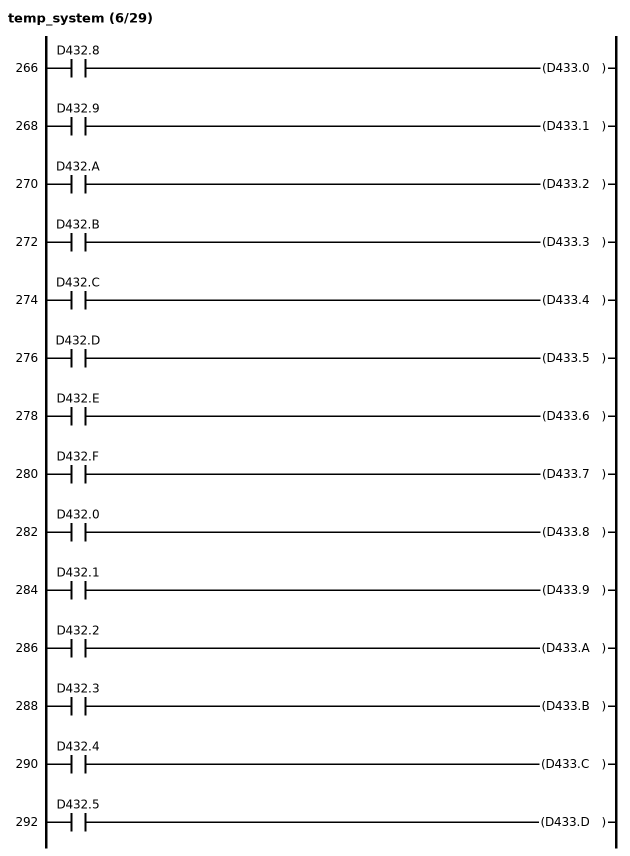
[picture p288: ladder of temp_system, rungs at steps 266 to 292]
266   LD      D432.8
      OUT     D433.0
268   LD      D432.9
      OUT     D433.1
270   LD      D432.A
      OUT     D433.2
272   LD      D432.B
      OUT     D433.3
274   LD      D432.C
      OUT     D433.4
276   LD      D432.D
      OUT     D433.5
278   LD      D432.E
      OUT     D433.6
280   LD      D432.F
      OUT     D433.7
282   LD      D432.0
      OUT     D433.8
284   LD      D432.1
      OUT     D433.9
286   LD      D432.2
      OUT     D433.A
288   LD      D432.3
      OUT     D433.B
290   LD      D432.4
      OUT     D433.C
292   LD      D432.5
      OUT     D433.D
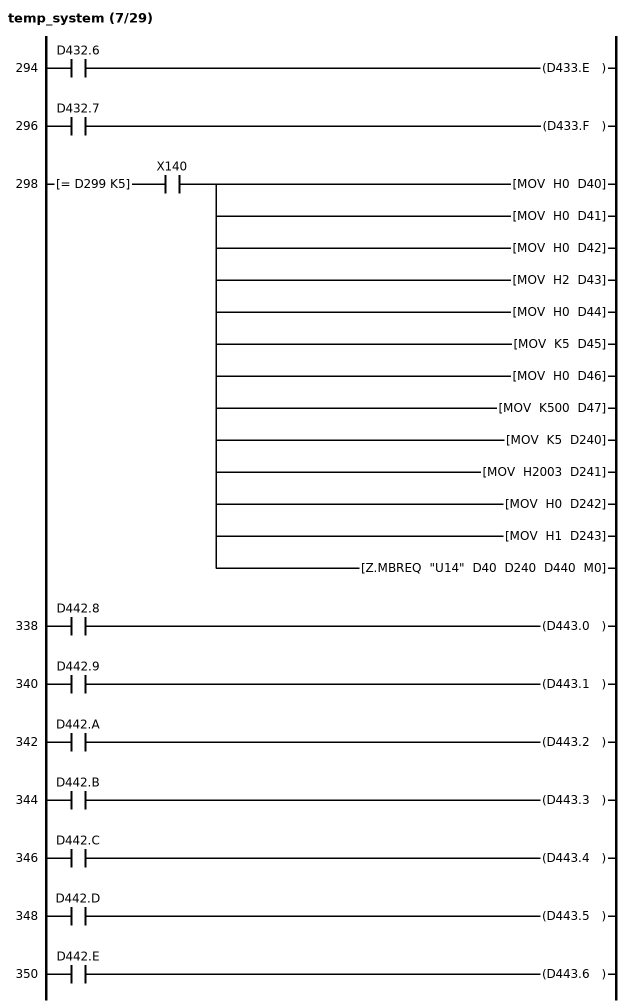
294   LD      D432.6
      OUT     D433.E
296   LD      D432.7
      OUT     D433.F
298   LD=     D299 K5
      AND     X140
      MOV     H0 D40
      MOV     H0 D41
      MOV     H0 D42
      MOV     H2 D43
      MOV     H0 D44
      MOV     K5 D45
      MOV     H0 D46
      MOV     K500 D47
      MOV     K5 D240
      MOV     H2003 D241
      MOV     H0 D242
      MOV     H1 D243
      Z.MBREQ "U14" D40 D240 D440 M0
338   LD      D442.8
      OUT     D443.0
340   LD      D442.9
      OUT     D443.1
342   LD      D442.A
      OUT     D443.2
344   LD      D442.B
      OUT     D443.3
346   LD      D442.C
      OUT     D443.4
348   LD      D442.D
      OUT     D443.5
350   LD      D442.E
      OUT     D443.6
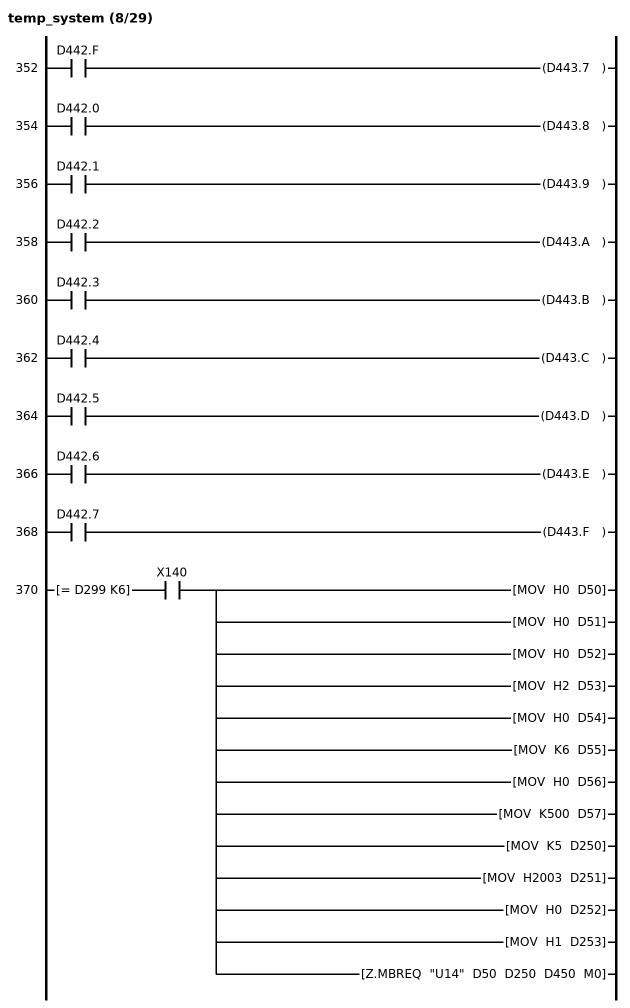
352   LD      D442.F
      OUT     D443.7
354   LD      D442.0
      OUT     D443.8
356   LD      D442.1
      OUT     D443.9
358   LD      D442.2
      OUT     D443.A
360   LD      D442.3
      OUT     D443.B
362   LD      D442.4
      OUT     D443.C
364   LD      D442.5
      OUT     D443.D
366   LD      D442.6
      OUT     D443.E
368   LD      D442.7
      OUT     D443.F
370   LD=     D299 K6
      AND     X140
      MOV     H0 D50
      MOV     H0 D51
      MOV     H0 D52
      MOV     H2 D53
      MOV     H0 D54
      MOV     K6 D55
      MOV     H0 D56
      MOV     K500 D57
      MOV     K5 D250
      MOV     H2003 D251
      MOV     H0 D252
      MOV     H1 D253
      Z.MBREQ "U14" D50 D250 D450 M0
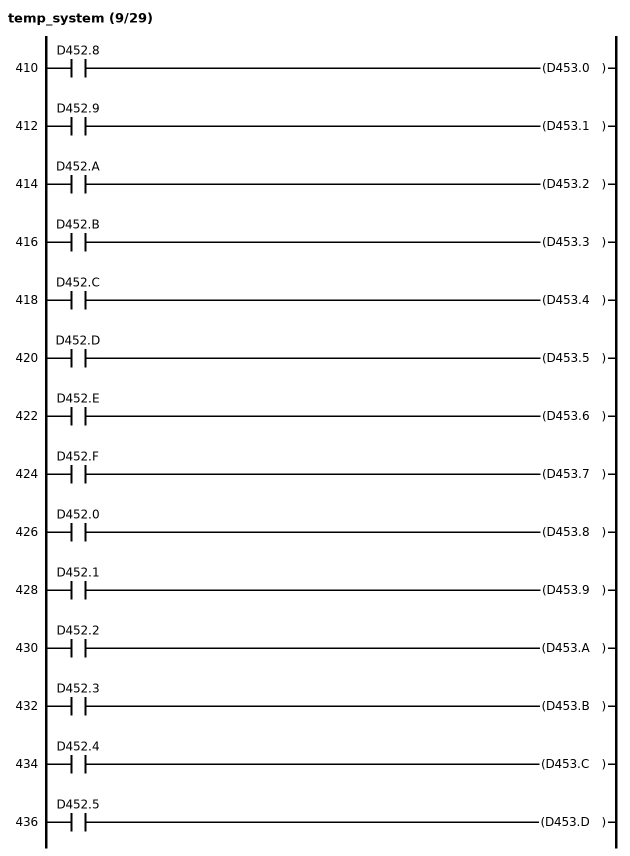
410   LD      D452.8
      OUT     D453.0
412   LD      D452.9
      OUT     D453.1
414   LD      D452.A
      OUT     D453.2
416   LD      D452.B
      OUT     D453.3
418   LD      D452.C
      OUT     D453.4
420   LD      D452.D
      OUT     D453.5
422   LD      D452.E
      OUT     D453.6
424   LD      D452.F
      OUT     D453.7
426   LD      D452.0
      OUT     D453.8
428   LD      D452.1
      OUT     D453.9
430   LD      D452.2
      OUT     D453.A
432   LD      D452.3
      OUT     D453.B
434   LD      D452.4
      OUT     D453.C
436   LD      D452.5
      OUT     D453.D
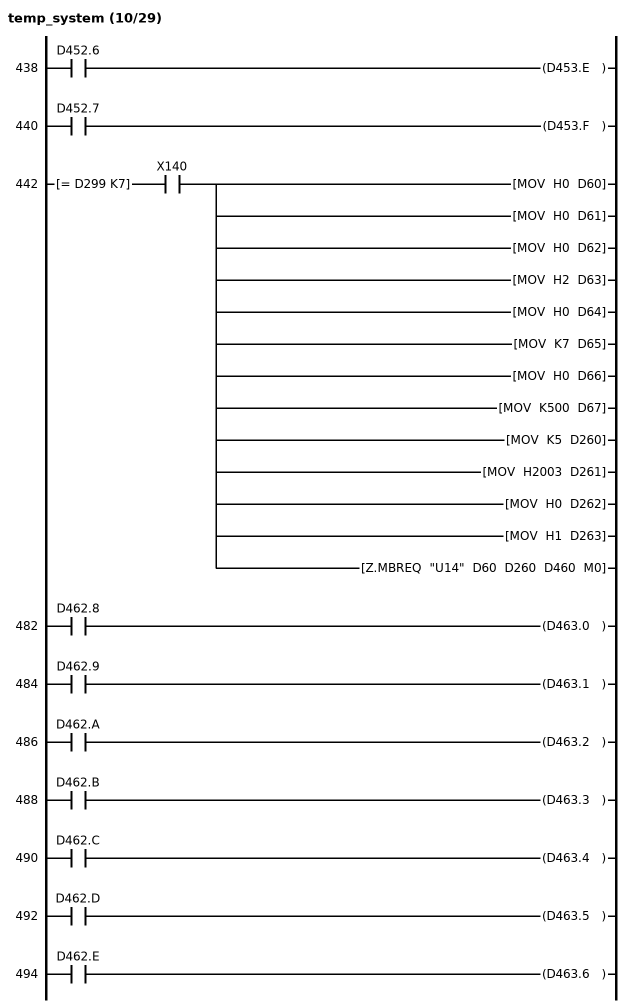
438   LD      D452.6
      OUT     D453.E
440   LD      D452.7
      OUT     D453.F
442   LD=     D299 K7
      AND     X140
      MOV     H0 D60
      MOV     H0 D61
      MOV     H0 D62
      MOV     H2 D63
      MOV     H0 D64
      MOV     K7 D65
      MOV     H0 D66
      MOV     K500 D67
      MOV     K5 D260
      MOV     H2003 D261
      MOV     H0 D262
      MOV     H1 D263
      Z.MBREQ "U14" D60 D260 D460 M0
482   LD      D462.8
      OUT     D463.0
484   LD      D462.9
      OUT     D463.1
486   LD      D462.A
      OUT     D463.2
488   LD      D462.B
      OUT     D463.3
490   LD      D462.C
      OUT     D463.4
492   LD      D462.D
      OUT     D463.5
494   LD      D462.E
      OUT     D463.6
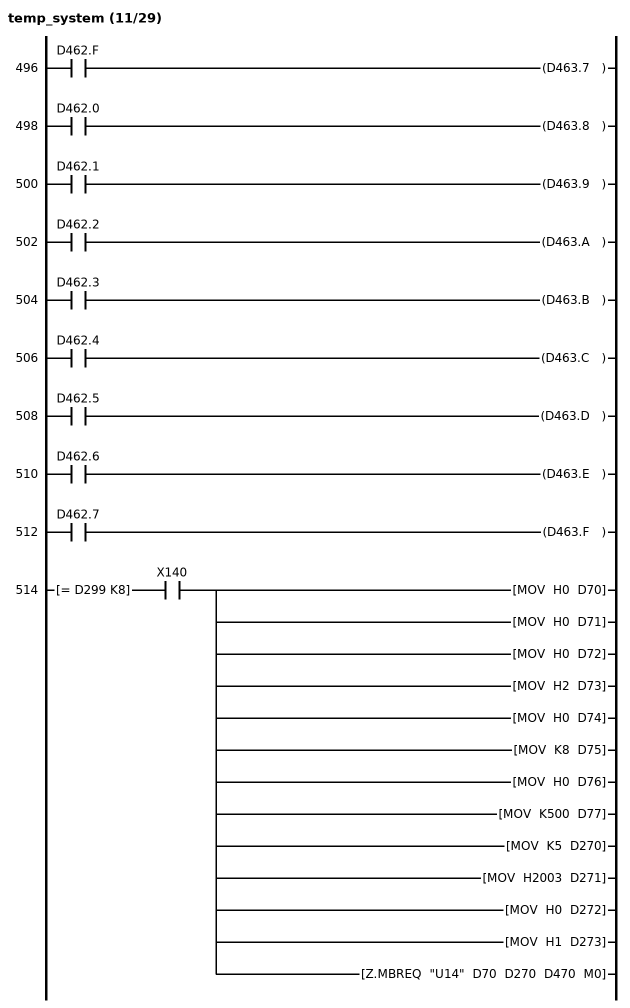
496   LD      D462.F
      OUT     D463.7
498   LD      D462.0
      OUT     D463.8
500   LD      D462.1
      OUT     D463.9
502   LD      D462.2
      OUT     D463.A
504   LD      D462.3
      OUT     D463.B
506   LD      D462.4
      OUT     D463.C
508   LD      D462.5
      OUT     D463.D
510   LD      D462.6
      OUT     D463.E
512   LD      D462.7
      OUT     D463.F
514   LD=     D299 K8
      AND     X140
      MOV     H0 D70
      MOV     H0 D71
      MOV     H0 D72
      MOV     H2 D73
      MOV     H0 D74
      MOV     K8 D75
      MOV     H0 D76
      MOV     K500 D77
      MOV     K5 D270
      MOV     H2003 D271
      MOV     H0 D272
      MOV     H1 D273
      Z.MBREQ "U14" D70 D270 D470 M0
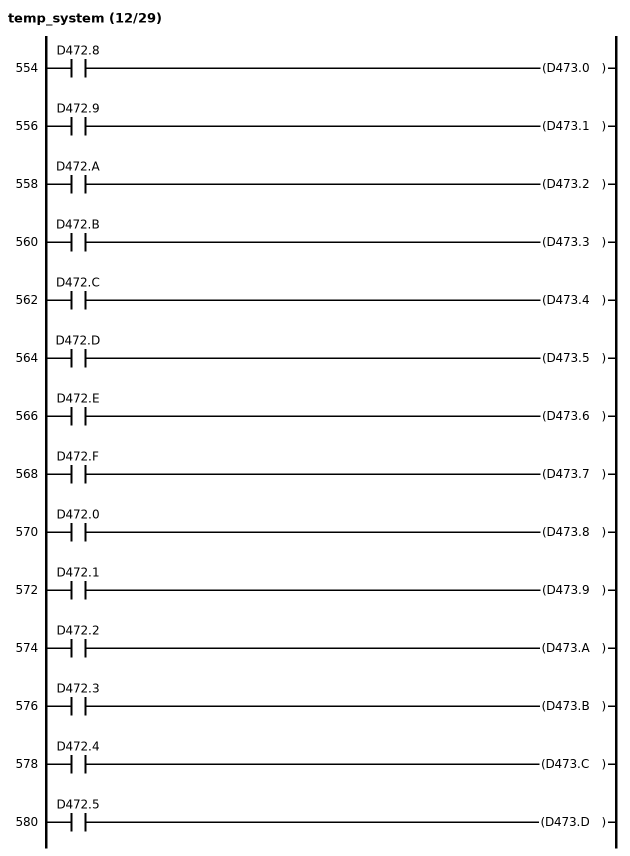
554   LD      D472.8
      OUT     D473.0
556   LD      D472.9
      OUT     D473.1
558   LD      D472.A
      OUT     D473.2
560   LD      D472.B
      OUT     D473.3
562   LD      D472.C
      OUT     D473.4
564   LD      D472.D
      OUT     D473.5
566   LD      D472.E
      OUT     D473.6
568   LD      D472.F
      OUT     D473.7
570   LD      D472.0
      OUT     D473.8
572   LD      D472.1
      OUT     D473.9
574   LD      D472.2
      OUT     D473.A
576   LD      D472.3
      OUT     D473.B
578   LD      D472.4
      OUT     D473.C
580   LD      D472.5
      OUT     D473.D
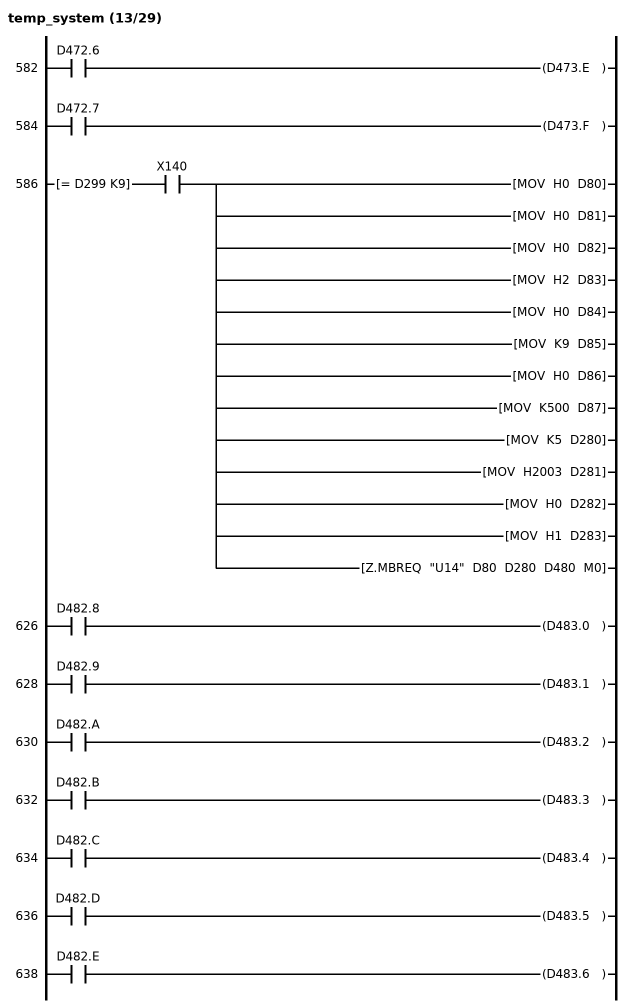
582   LD      D472.6
      OUT     D473.E
584   LD      D472.7
      OUT     D473.F
586   LD=     D299 K9
      AND     X140
      MOV     H0 D80
      MOV     H0 D81
      MOV     H0 D82
      MOV     H2 D83
      MOV     H0 D84
      MOV     K9 D85
      MOV     H0 D86
      MOV     K500 D87
      MOV     K5 D280
      MOV     H2003 D281
      MOV     H0 D282
      MOV     H1 D283
      Z.MBREQ "U14" D80 D280 D480 M0
626   LD      D482.8
      OUT     D483.0
628   LD      D482.9
      OUT     D483.1
630   LD      D482.A
      OUT     D483.2
632   LD      D482.B
      OUT     D483.3
634   LD      D482.C
      OUT     D483.4
636   LD      D482.D
      OUT     D483.5
638   LD      D482.E
      OUT     D483.6
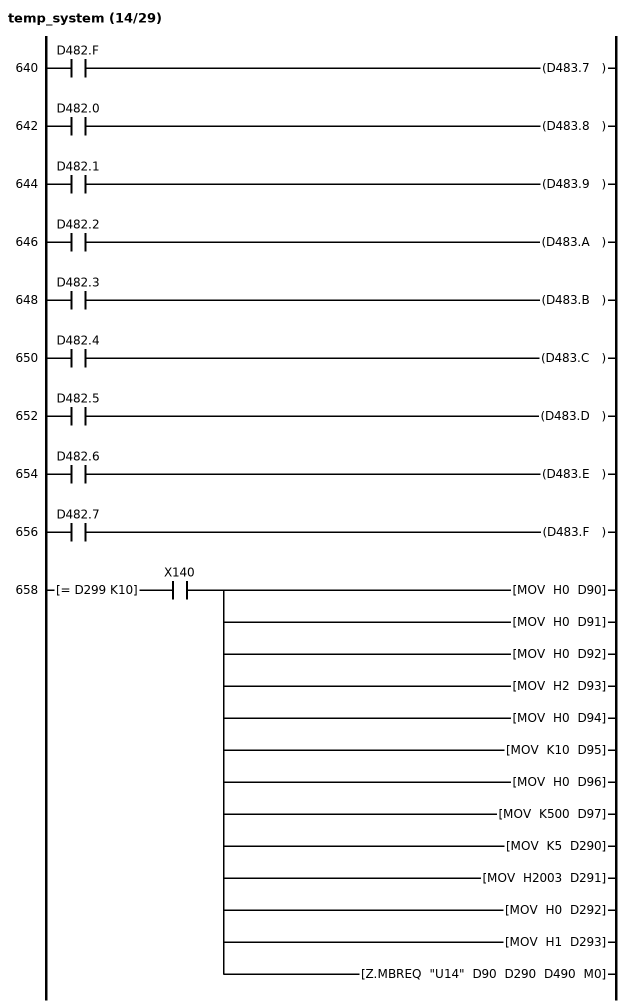
640   LD      D482.F
      OUT     D483.7
642   LD      D482.0
      OUT     D483.8
644   LD      D482.1
      OUT     D483.9
646   LD      D482.2
      OUT     D483.A
648   LD      D482.3
      OUT     D483.B
650   LD      D482.4
      OUT     D483.C
652   LD      D482.5
      OUT     D483.D
654   LD      D482.6
      OUT     D483.E
656   LD      D482.7
      OUT     D483.F
658   LD=     D299 K10
      AND     X140
      MOV     H0 D90
      MOV     H0 D91
      MOV     H0 D92
      MOV     H2 D93
      MOV     H0 D94
      MOV     K10 D95
      MOV     H0 D96
      MOV     K500 D97
      MOV     K5 D290
      MOV     H2003 D291
      MOV     H0 D292
      MOV     H1 D293
      Z.MBREQ "U14" D90 D290 D490 M0
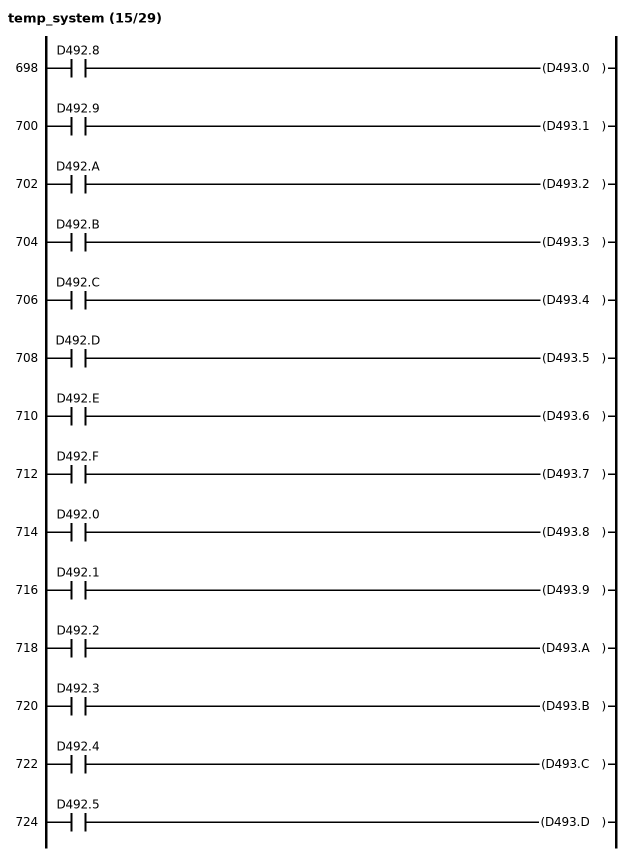
698   LD      D492.8
      OUT     D493.0
700   LD      D492.9
      OUT     D493.1
702   LD      D492.A
      OUT     D493.2
704   LD      D492.B
      OUT     D493.3
706   LD      D492.C
      OUT     D493.4
708   LD      D492.D
      OUT     D493.5
710   LD      D492.E
      OUT     D493.6
712   LD      D492.F
      OUT     D493.7
714   LD      D492.0
      OUT     D493.8
716   LD      D492.1
      OUT     D493.9
718   LD      D492.2
      OUT     D493.A
720   LD      D492.3
      OUT     D493.B
722   LD      D492.4
      OUT     D493.C
724   LD      D492.5
      OUT     D493.D
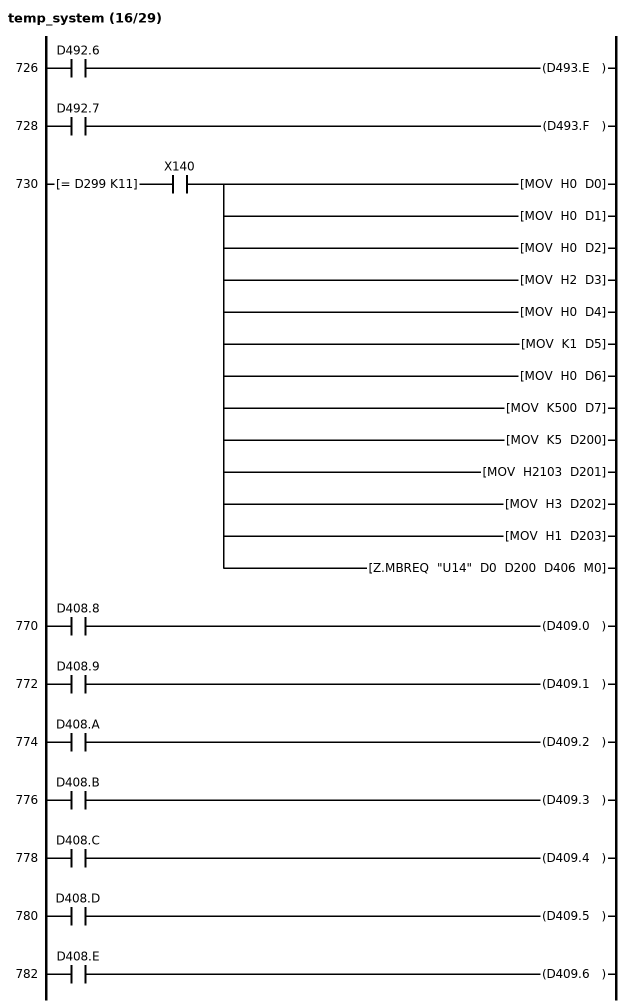
726   LD      D492.6
      OUT     D493.E
728   LD      D492.7
      OUT     D493.F
730   LD=     D299 K11
      AND     X140
      MOV     H0 D0
      MOV     H0 D1
      MOV     H0 D2
      MOV     H2 D3
      MOV     H0 D4
      MOV     K1 D5
      MOV     H0 D6
      MOV     K500 D7
      MOV     K5 D200
      MOV     H2103 D201
      MOV     H3 D202
      MOV     H1 D203
      Z.MBREQ "U14" D0 D200 D406 M0
770   LD      D408.8
      OUT     D409.0
772   LD      D408.9
      OUT     D409.1
774   LD      D408.A
      OUT     D409.2
776   LD      D408.B
      OUT     D409.3
778   LD      D408.C
      OUT     D409.4
780   LD      D408.D
      OUT     D409.5
782   LD      D408.E
      OUT     D409.6
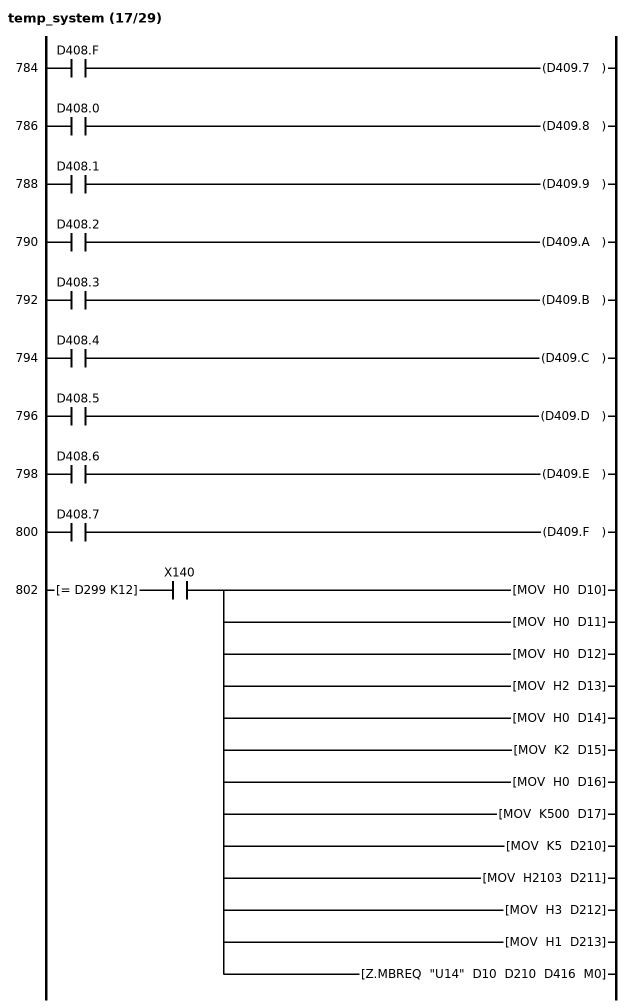
784   LD      D408.F
      OUT     D409.7
786   LD      D408.0
      OUT     D409.8
788   LD      D408.1
      OUT     D409.9
790   LD      D408.2
      OUT     D409.A
792   LD      D408.3
      OUT     D409.B
794   LD      D408.4
      OUT     D409.C
796   LD      D408.5
      OUT     D409.D
798   LD      D408.6
      OUT     D409.E
800   LD      D408.7
      OUT     D409.F
802   LD=     D299 K12
      AND     X140
      MOV     H0 D10
      MOV     H0 D11
      MOV     H0 D12
      MOV     H2 D13
      MOV     H0 D14
      MOV     K2 D15
      MOV     H0 D16
      MOV     K500 D17
      MOV     K5 D210
      MOV     H2103 D211
      MOV     H3 D212
      MOV     H1 D213
      Z.MBREQ "U14" D10 D210 D416 M0
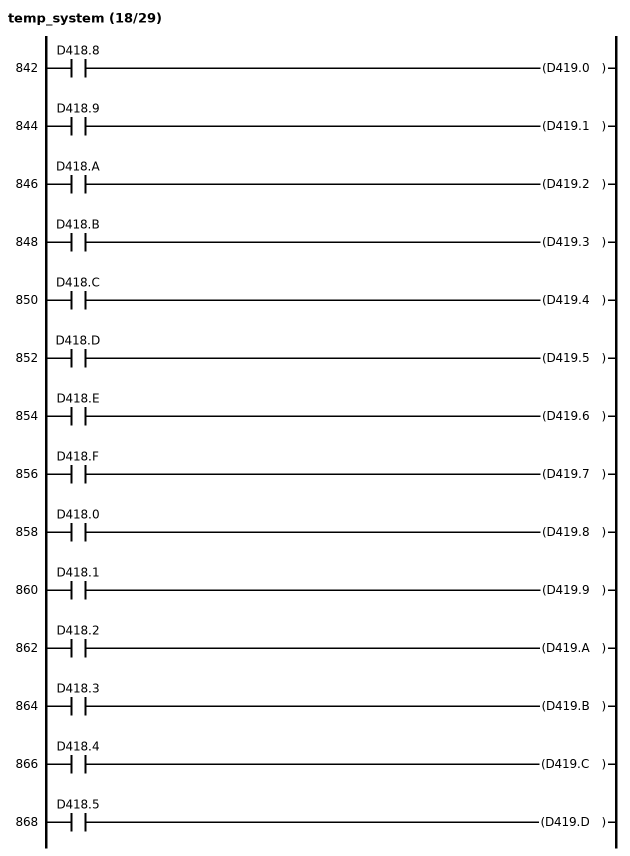
842   LD      D418.8
      OUT     D419.0
844   LD      D418.9
      OUT     D419.1
846   LD      D418.A
      OUT     D419.2
848   LD      D418.B
      OUT     D419.3
850   LD      D418.C
      OUT     D419.4
852   LD      D418.D
      OUT     D419.5
854   LD      D418.E
      OUT     D419.6
856   LD      D418.F
      OUT     D419.7
858   LD      D418.0
      OUT     D419.8
860   LD      D418.1
      OUT     D419.9
862   LD      D418.2
      OUT     D419.A
864   LD      D418.3
      OUT     D419.B
866   LD      D418.4
      OUT     D419.C
868   LD      D418.5
      OUT     D419.D
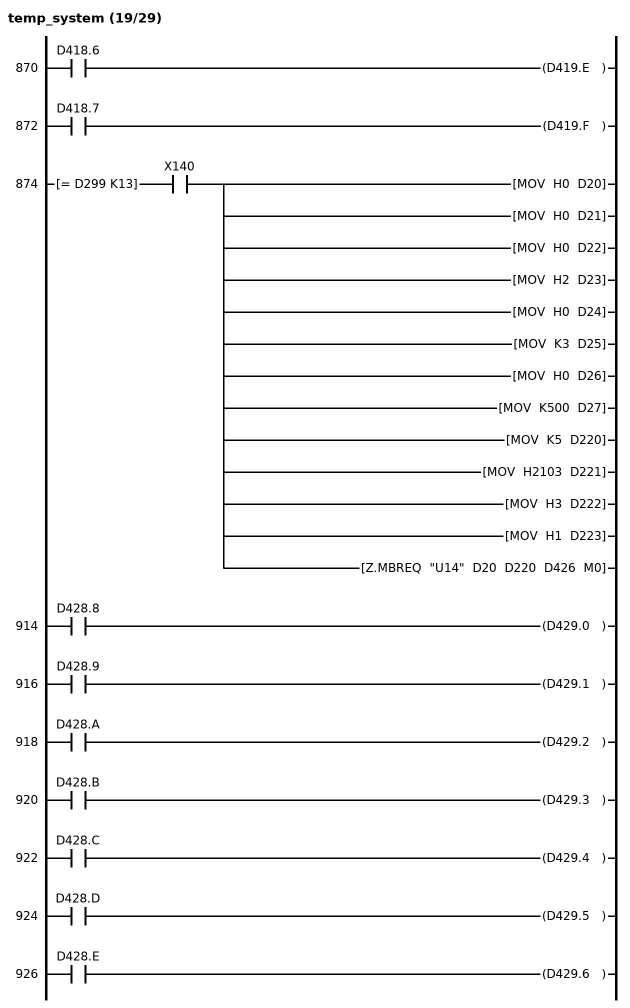
870   LD      D418.6
      OUT     D419.E
872   LD      D418.7
      OUT     D419.F
874   LD=     D299 K13
      AND     X140
      MOV     H0 D20
      MOV     H0 D21
      MOV     H0 D22
      MOV     H2 D23
      MOV     H0 D24
      MOV     K3 D25
      MOV     H0 D26
      MOV     K500 D27
      MOV     K5 D220
      MOV     H2103 D221
      MOV     H3 D222
      MOV     H1 D223
      Z.MBREQ "U14" D20 D220 D426 M0
914   LD      D428.8
      OUT     D429.0
916   LD      D428.9
      OUT     D429.1
918   LD      D428.A
      OUT     D429.2
920   LD      D428.B
      OUT     D429.3
922   LD      D428.C
      OUT     D429.4
924   LD      D428.D
      OUT     D429.5
926   LD      D428.E
      OUT     D429.6
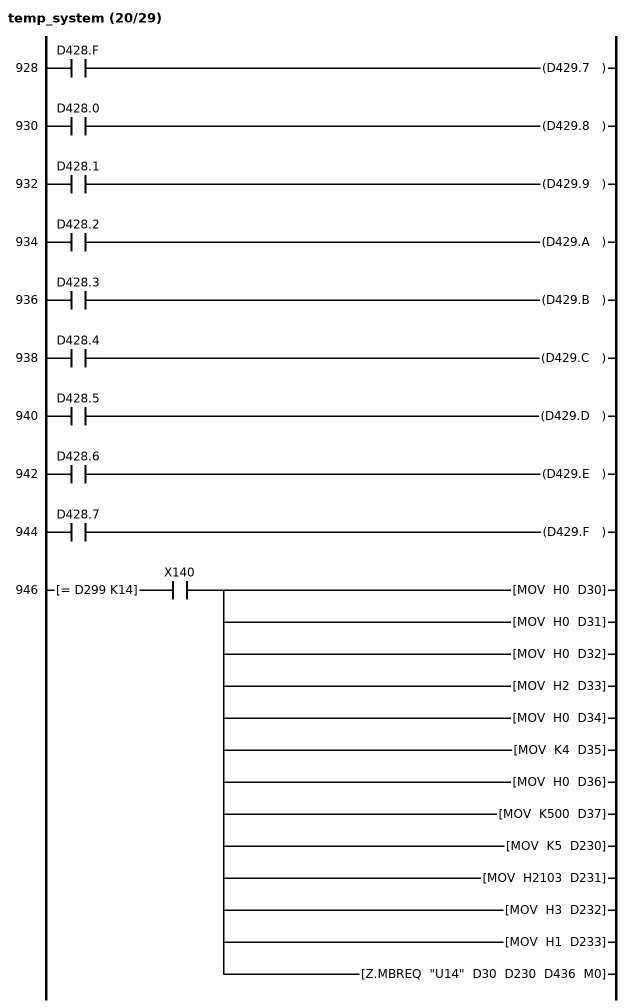
928   LD      D428.F
      OUT     D429.7
930   LD      D428.0
      OUT     D429.8
932   LD      D428.1
      OUT     D429.9
934   LD      D428.2
      OUT     D429.A
936   LD      D428.3
      OUT     D429.B
938   LD      D428.4
      OUT     D429.C
940   LD      D428.5
      OUT     D429.D
942   LD      D428.6
      OUT     D429.E
944   LD      D428.7
      OUT     D429.F
946   LD=     D299 K14
      AND     X140
      MOV     H0 D30
      MOV     H0 D31
      MOV     H0 D32
      MOV     H2 D33
      MOV     H0 D34
      MOV     K4 D35
      MOV     H0 D36
      MOV     K500 D37
      MOV     K5 D230
      MOV     H2103 D231
      MOV     H3 D232
      MOV     H1 D233
      Z.MBREQ "U14" D30 D230 D436 M0
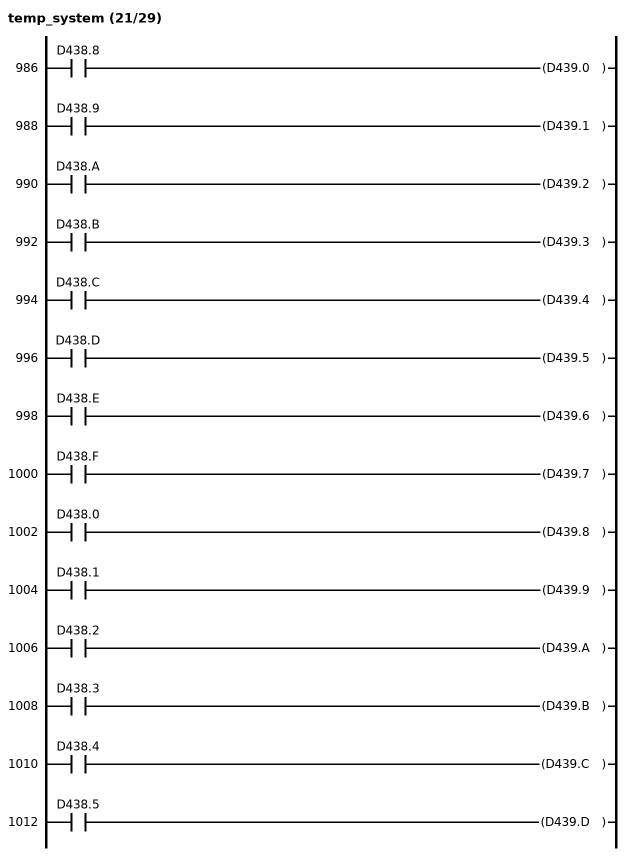
986   LD      D438.8
      OUT     D439.0
988   LD      D438.9
      OUT     D439.1
990   LD      D438.A
      OUT     D439.2
992   LD      D438.B
      OUT     D439.3
994   LD      D438.C
      OUT     D439.4
996   LD      D438.D
      OUT     D439.5
998   LD      D438.E
      OUT     D439.6
1000  LD      D438.F
      OUT     D439.7
1002  LD      D438.0
      OUT     D439.8
1004  LD      D438.1
      OUT     D439.9
1006  LD      D438.2
      OUT     D439.A
1008  LD      D438.3
      OUT     D439.B
1010  LD      D438.4
      OUT     D439.C
1012  LD      D438.5
      OUT     D439.D
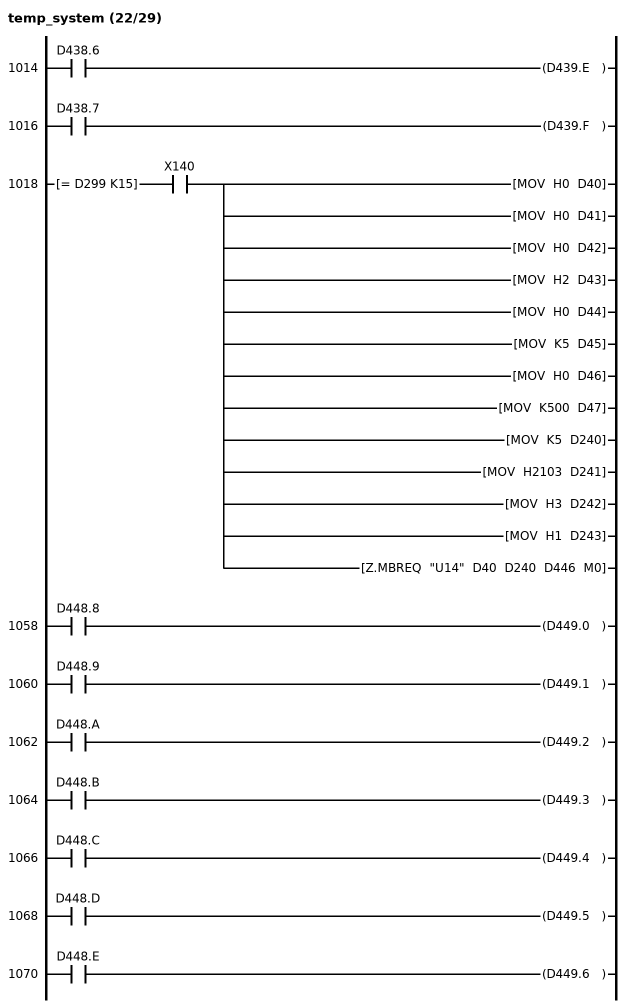
1014  LD      D438.6
      OUT     D439.E
1016  LD      D438.7
      OUT     D439.F
1018  LD=     D299 K15
      AND     X140
      MOV     H0 D40
      MOV     H0 D41
      MOV     H0 D42
      MOV     H2 D43
      MOV     H0 D44
      MOV     K5 D45
      MOV     H0 D46
      MOV     K500 D47
      MOV     K5 D240
      MOV     H2103 D241
      MOV     H3 D242
      MOV     H1 D243
      Z.MBREQ "U14" D40 D240 D446 M0
1058  LD      D448.8
      OUT     D449.0
1060  LD      D448.9
      OUT     D449.1
1062  LD      D448.A
      OUT     D449.2
1064  LD      D448.B
      OUT     D449.3
1066  LD      D448.C
      OUT     D449.4
1068  LD      D448.D
      OUT     D449.5
1070  LD      D448.E
      OUT     D449.6
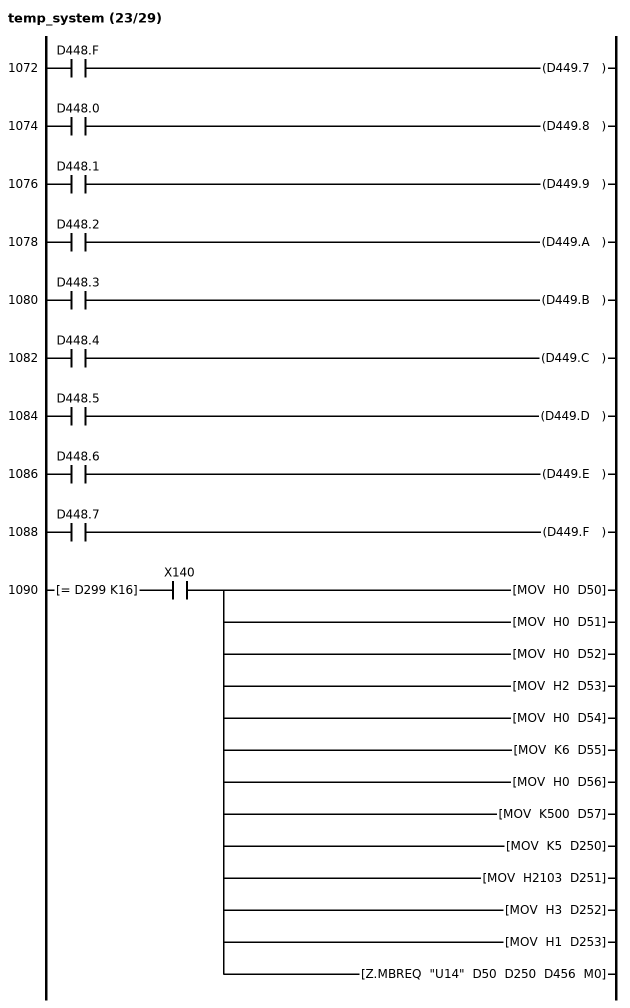
1072  LD      D448.F
      OUT     D449.7
1074  LD      D448.0
      OUT     D449.8
1076  LD      D448.1
      OUT     D449.9
1078  LD      D448.2
      OUT     D449.A
1080  LD      D448.3
      OUT     D449.B
1082  LD      D448.4
      OUT     D449.C
1084  LD      D448.5
      OUT     D449.D
1086  LD      D448.6
      OUT     D449.E
1088  LD      D448.7
      OUT     D449.F
1090  LD=     D299 K16
      AND     X140
      MOV     H0 D50
      MOV     H0 D51
      MOV     H0 D52
      MOV     H2 D53
      MOV     H0 D54
      MOV     K6 D55
      MOV     H0 D56
      MOV     K500 D57
      MOV     K5 D250
      MOV     H2103 D251
      MOV     H3 D252
      MOV     H1 D253
      Z.MBREQ "U14" D50 D250 D456 M0
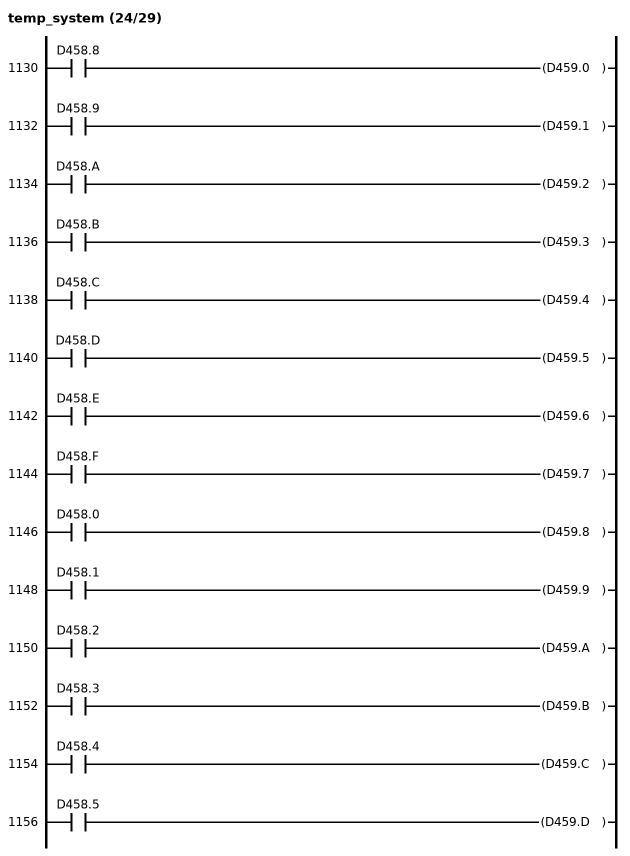
1130  LD      D458.8
      OUT     D459.0
1132  LD      D458.9
      OUT     D459.1
1134  LD      D458.A
      OUT     D459.2
1136  LD      D458.B
      OUT     D459.3
1138  LD      D458.C
      OUT     D459.4
1140  LD      D458.D
      OUT     D459.5
1142  LD      D458.E
      OUT     D459.6
1144  LD      D458.F
      OUT     D459.7
1146  LD      D458.0
      OUT     D459.8
1148  LD      D458.1
      OUT     D459.9
1150  LD      D458.2
      OUT     D459.A
1152  LD      D458.3
      OUT     D459.B
1154  LD      D458.4
      OUT     D459.C
1156  LD      D458.5
      OUT     D459.D
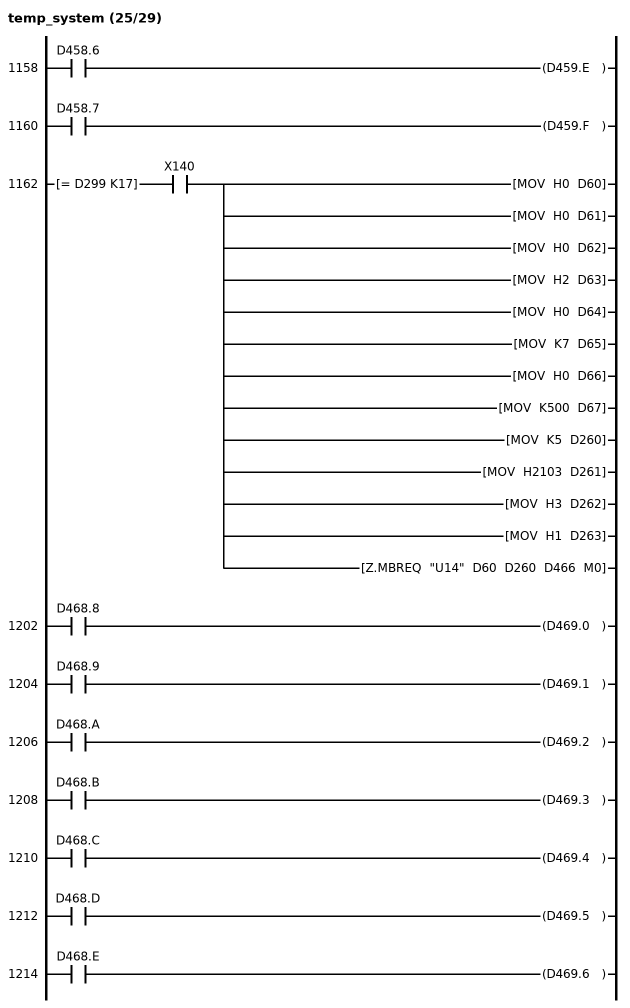
1158  LD      D458.6
      OUT     D459.E
1160  LD      D458.7
      OUT     D459.F
1162  LD=     D299 K17
      AND     X140
      MOV     H0 D60
      MOV     H0 D61
      MOV     H0 D62
      MOV     H2 D63
      MOV     H0 D64
      MOV     K7 D65
      MOV     H0 D66
      MOV     K500 D67
      MOV     K5 D260
      MOV     H2103 D261
      MOV     H3 D262
      MOV     H1 D263
      Z.MBREQ "U14" D60 D260 D466 M0
1202  LD      D468.8
      OUT     D469.0
1204  LD      D468.9
      OUT     D469.1
1206  LD      D468.A
      OUT     D469.2
1208  LD      D468.B
      OUT     D469.3
1210  LD      D468.C
      OUT     D469.4
1212  LD      D468.D
      OUT     D469.5
1214  LD      D468.E
      OUT     D469.6
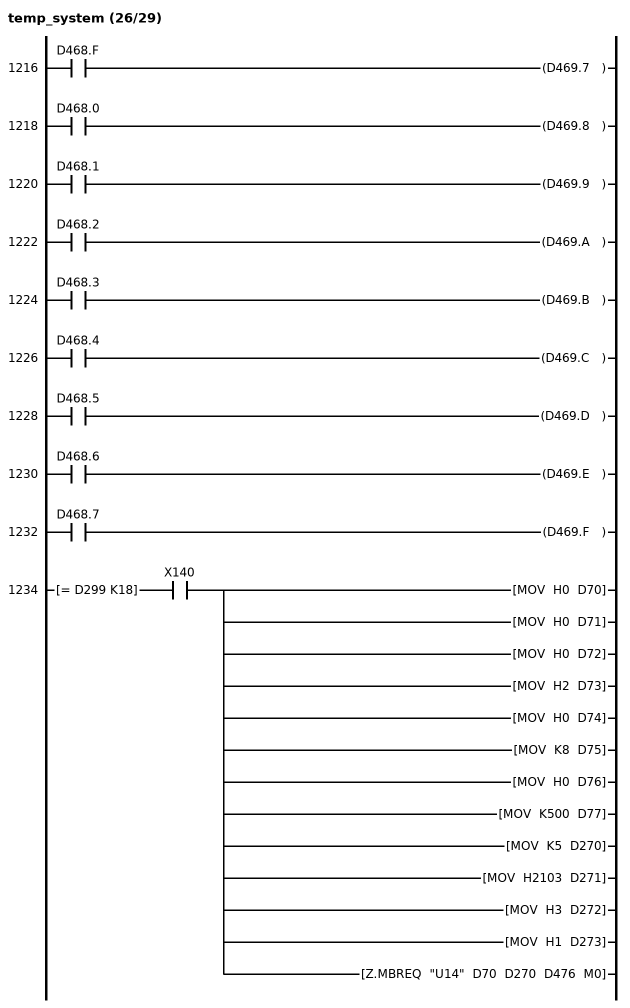
1216  LD      D468.F
      OUT     D469.7
1218  LD      D468.0
      OUT     D469.8
1220  LD      D468.1
      OUT     D469.9
1222  LD      D468.2
      OUT     D469.A
1224  LD      D468.3
      OUT     D469.B
1226  LD      D468.4
      OUT     D469.C
1228  LD      D468.5
      OUT     D469.D
1230  LD      D468.6
      OUT     D469.E
1232  LD      D468.7
      OUT     D469.F
1234  LD=     D299 K18
      AND     X140
      MOV     H0 D70
      MOV     H0 D71
      MOV     H0 D72
      MOV     H2 D73
      MOV     H0 D74
      MOV     K8 D75
      MOV     H0 D76
      MOV     K500 D77
      MOV     K5 D270
      MOV     H2103 D271
      MOV     H3 D272
      MOV     H1 D273
      Z.MBREQ "U14" D70 D270 D476 M0
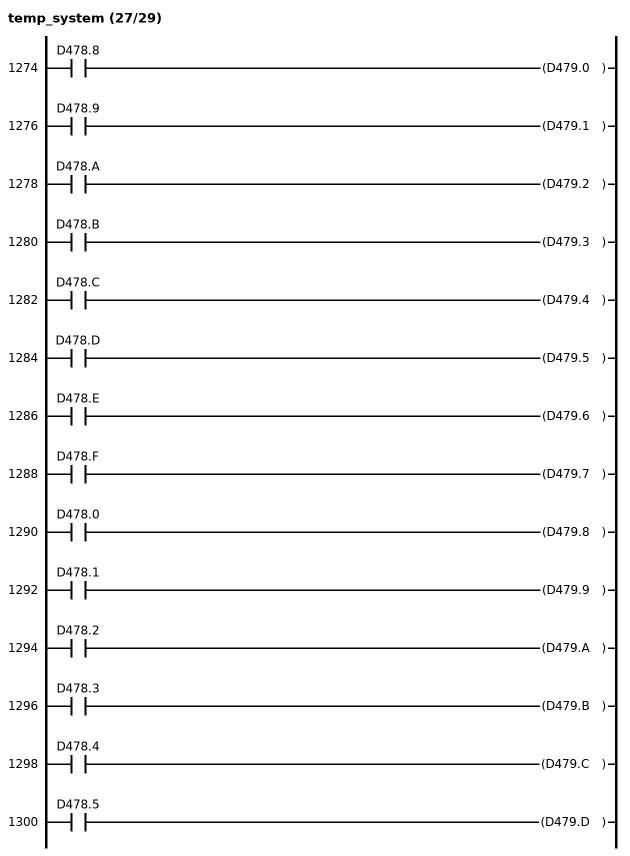
1274  LD      D478.8
      OUT     D479.0
1276  LD      D478.9
      OUT     D479.1
1278  LD      D478.A
      OUT     D479.2
1280  LD      D478.B
      OUT     D479.3
1282  LD      D478.C
      OUT     D479.4
1284  LD      D478.D
      OUT     D479.5
1286  LD      D478.E
      OUT     D479.6
1288  LD      D478.F
      OUT     D479.7
1290  LD      D478.0
      OUT     D479.8
1292  LD      D478.1
      OUT     D479.9
1294  LD      D478.2
      OUT     D479.A
1296  LD      D478.3
      OUT     D479.B
1298  LD      D478.4
      OUT     D479.C
1300  LD      D478.5
      OUT     D479.D
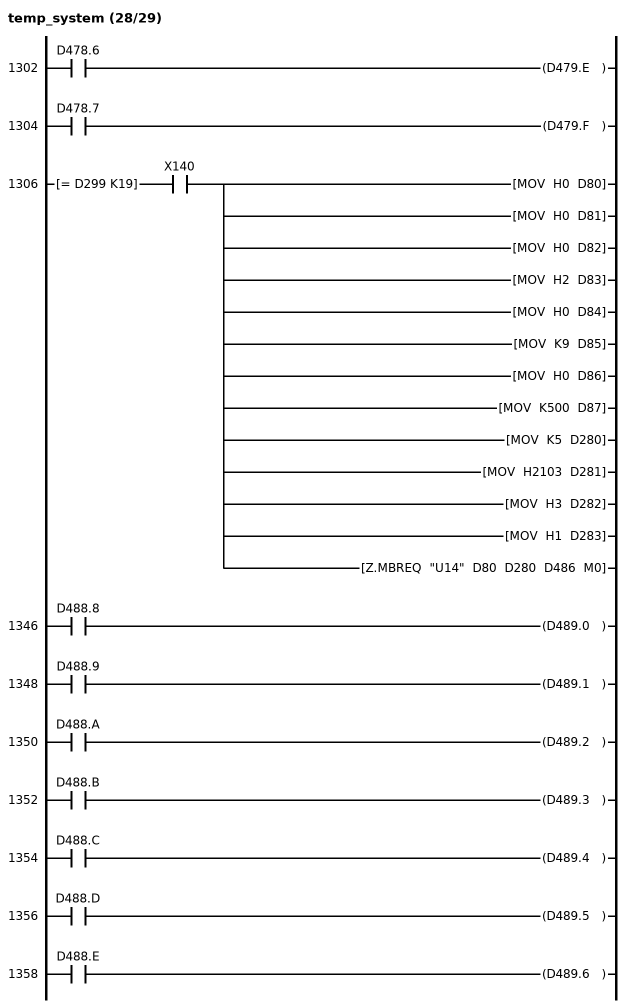
1302  LD      D478.6
      OUT     D479.E
1304  LD      D478.7
      OUT     D479.F
1306  LD=     D299 K19
      AND     X140
      MOV     H0 D80
      MOV     H0 D81
      MOV     H0 D82
      MOV     H2 D83
      MOV     H0 D84
      MOV     K9 D85
      MOV     H0 D86
      MOV     K500 D87
      MOV     K5 D280
      MOV     H2103 D281
      MOV     H3 D282
      MOV     H1 D283
      Z.MBREQ "U14" D80 D280 D486 M0
1346  LD      D488.8
      OUT     D489.0
1348  LD      D488.9
      OUT     D489.1
1350  LD      D488.A
      OUT     D489.2
1352  LD      D488.B
      OUT     D489.3
1354  LD      D488.C
      OUT     D489.4
1356  LD      D488.D
      OUT     D489.5
1358  LD      D488.E
      OUT     D489.6
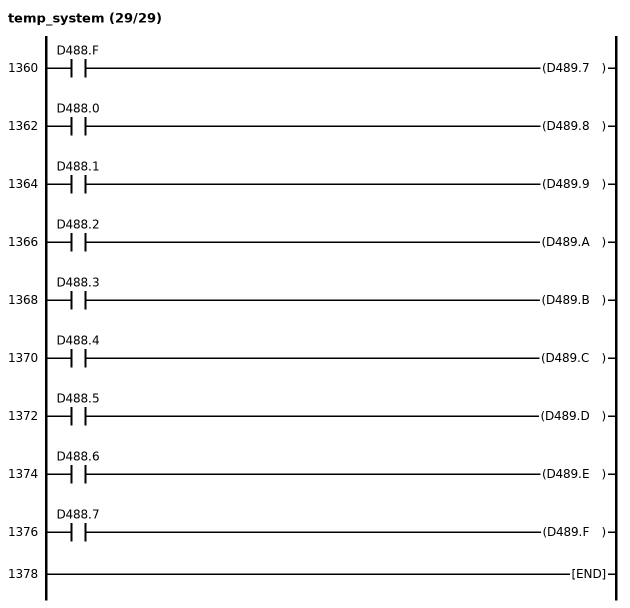
1360  LD      D488.F
      OUT     D489.7
1362  LD      D488.0
      OUT     D489.8
1364  LD      D488.1
      OUT     D489.9
1366  LD      D488.2
      OUT     D489.A
1368  LD      D488.3
      OUT     D489.B
1370  LD      D488.4
      OUT     D489.C
1372  LD      D488.5
      OUT     D489.D
1374  LD      D488.6
      OUT     D489.E
1376  LD      D488.7
      OUT     D489.F
1378  END
END_PROGRAM

PROGRAM tower_lamp
